Staubli VAL3: SetDrivePwrMsg.dtx

public Body body
  [0]
    num nData
public Header header
  [0]
    num nCommType
    num nData[12]
    num nMsgType
    num nReplyCode
public Prefix prefix
  [0]
    num nData[4]
    num nLength
public bool bDrivePower
